SUBAPPLICATION IXA_TO_logiBUS_LED_strip_QXA (* Taster IXA schaltet einen LED-Strip blinkend (Farbe, Strip-Nummer parametrierbar), adapter-basiert. Generisch. Schwester-Baustein zu MyLib::sys::IX_TO_logiBUS_LED_strip_QX (dort event-basiert statt AX-Adapter). *)
  (* Standard: 61499-2 *)
  (* Version 1.1, 2026-09-18, Franz Höpfinger, Meisterschulen am Ostbahnhof, BUTTON.INITO auf BUTTON.REQ zurueckverdrahtet (Selfloop) - loest nach der Initialisierung sofort einen Service-Request aus, statt auf die erste echte Wertaenderung am Bus zu warten (Fix fuer 'Waiting for handle'-Status direkt nach Boot). *)
  (* Version 1.0, 2026-09-09, Franz Höpfinger, Meisterschulen am Ostbahnhof, Angelegt beim Portieren von Uebung_033 nach test_AX zur Wiederverwendung. *)
  PACKAGE MyLib::sys;
  IMPORT logiBUS::io::DI::logiBUS_DI_S;
  IMPORT logiBUS::io::DO_LED::LED_COLOURS;
  IMPORT logiBUS::io::DO_LED::LED_FREQ;
  IMPORT logiBUS::io::DI::logiBUS_DI::Invalid;
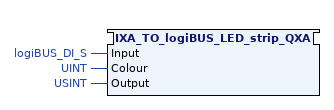
  VAR_INPUT
    Input : logiBUS::io::DI::logiBUS_DI_S := Invalid; (* Identify the Input Input_I1..I8 *)
    Colour : UINT := LED_COLOURS::LED_GREEN; (* This identify the Colour. *)
    Output : USINT; (* Identify the Output Number of Strip *)
  END_VAR
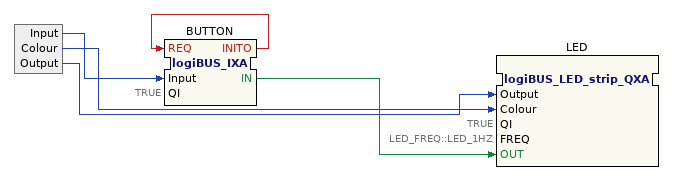
  FBS
    LED : logiBUS::io::DO_LED::logiBUS_LED_strip_QXA(QI := TRUE, FREQ := LED_FREQ::LED_1HZ);
    BUTTON : logiBUS::io::DI::logiBUS_IXA(QI := TRUE);
  END_FBS
  EVENT_CONNECTIONS
    BUTTON.INITO TO BUTTON.REQ;
  END_CONNECTIONS
  DATA_CONNECTIONS
    Input TO BUTTON.Input;
    Output TO LED.Output;
    Colour TO LED.Colour;
  END_CONNECTIONS
  ADAPTER_CONNECTIONS
    BUTTON.IN TO LED.OUT;
  END_CONNECTIONS
END_SUBAPPLICATION
